(* IEC 61131-3 sources: repolevel_ST_code_completion/output/0127完整版本_带planner/repoeval_plc_hello_mixing_tank/readful_result_no_provide, 5 files *)

(* ---- F_ResetDeviceCommands.st ---- *)
VAR
	bAllCommandsReset : BOOL := TRUE;
END_VAR

// 混合电机命令复位
IF bMixerRunning THEN
	bMixerRunCmd := FALSE;
	bMixerStopCmd := FALSE;
ELSE
	bAllCommandsReset := FALSE;
END_IF

// 介质1阀门命令复位
IF bMedium1Opened THEN
	bMedium1OpenCmd := FALSE;
	bMedium1CloseCmd := FALSE;
ELSE
	bAllCommandsReset := FALSE;
END_IF

// 介质2阀门命令复位
IF bMedium2Opened THEN
	bMedium2OpenCmd := FALSE;
	bMedium2CloseCmd := FALSE;
ELSE
	bAllCommandsReset := FALSE;
END_IF

// 排水阀门命令复位
IF bDrainOpened THEN
	bDrainOpenCmd := FALSE;
	bDrainCloseCmd := FALSE;
ELSE
	bAllCommandsReset := FALSE;
END_IF

// 返回所有命令是否已复位
F_ResetDeviceCommands := bAllCommandsReset;
RETURN;
END_FUNCTION

(* ---- F_UpdateLimitSwitches.st ---- *)
bLevelFull := rTankLevel >= rFullThreshold;
bLevelEmpty := rTankLevel <= rEmptyThreshold;
F_UpdateLimitSwitches := TRUE;
RETURN;
END_FUNCTION

(* ---- FB_AutoSequence.st ---- *)
VAR
	tonMixing			:	TON;			// 混合定时器
END_VAR

// 初始化设备控制输出
bMixerRunCmd := FALSE;
bMedium1OpenCmd := FALSE;
bMedium2OpenCmd := FALSE;
bDrainOpenCmd := FALSE;

// 检查复位条件
IF bReset THEN
// Replace AUTO_SEQUENCE.DRAINING with a constant value or default state
  eCurrentState := 0; // Assuming '0' corresponds to the DRAINING state
	nCyclesCompleted := 0;
	RETURN;
END_IF

// 检查使能条件
IF NOT bEnable THEN
// Replace AUTO_SEQUENCE.IDLE with a constant value or default state
  eCurrentState := 1; // Assuming '1' corresponds to the IDLE state
	RETURN;
END_IF

// 自动序列状态机
CASE eCurrentState OF
0:	// DRAINING state
 // 排空状态逻辑
 bDrainOpenCmd := TRUE;
 IF bTankLevelEmpty THEN
 eCurrentState := 2; // Transition to FILLING state
 END_IF;

2:	// FILLING state
 // 填充状态逻辑
 bMedium1OpenCmd := TRUE;
 bMedium2OpenCmd := TRUE;
 IF bTankLevelFull THEN
 eCurrentState := 3; // Transition to MIXING state
 END_IF;

3:	// MIXING state
 // 混合状态逻辑
 bMixerRunCmd := TRUE;
 tonMixing(IN := TRUE, PT := tMixingDuration);
 IF tonMixing.Q THEN
 eCurrentState := 0; // Transition back to DRAINING state
 nCyclesCompleted := nCyclesCompleted + 1;
 END_IF;

ELSE
 // 默认状态为初始状态
 eCurrentState := 1; // IDLE state
END_CASE
END_FUNCTION_BLOCK

(* ---- FB_ManualControl.st ---- *)
bMixerRunCmdOut := (bMixerRunCmd OR bMixerRunning) AND NOT bMixerStopCmd;

bMedium1OpenCmdOut := (bMedium1OpenCmd OR bMedium1Opened) AND NOT bMedium1CloseCmd;

bMedium2OpenCmdOut := (bMedium2OpenCmd OR bMedium2Opened) AND NOT bMedium2CloseCmd;

bDrainOpenCmdOut := (bDrainOpenCmd OR bDrainOpened) AND NOT bDrainCloseCmd;
END_FUNCTION_BLOCK

(* ---- FB_TankLevelSimulator.st ---- *)
VAR
	rTempLevel : REAL; // 临时变量用于液位计算
END_VAR

// 复位逻辑
IF bReset THEN
	rCurrentLevel := rInitialLevel;
ELSE
	// 液位计算
	rTempLevel := rCurrentLevel
				+ rFillRate1 * BOOL_TO_REAL(bMedium1Opened)
				+ rFillRate2 * BOOL_TO_REAL(bMedium2Opened)
				- rDrainRate * BOOL_TO_REAL(bDrainOpened);

	// 边界检查
	IF rTempLevel > rMaxLevel THEN
		rCurrentLevel := rMaxLevel;
	ELSIF rTempLevel < rMinLevel THEN
		rCurrentLevel := rMinLevel;
	ELSE
		rCurrentLevel := rTempLevel;
	END_IF;
END_IF;
END_FUNCTION_BLOCK
